# EPICS autosave request: iocBoot/ioc2/dbSave/23i_CS_Av_.req
%
% BURT Request File
%
% 23i:CS:Av:  Collimator (Monochromatic) slits, Vertical Aperture
%

file $(DIR)/assy.req ASSY=23i:CS:Av
23i:CS:Av:Invert
file $(DIR)/mtr1.req MTR1=23i:CS:mz1
file $(DIR)/mtr1.req MTR1=23i:CS:mz2
file $(DIR)/drv1.req DRV1=23i:CS:ZT
file $(DIR)/drv1.req DRV1=23i:CS:ZB
file $(DIR)/axs1.req AXS1=23i:CS:ZC
file $(DIR)/axs1.req AXS1=23i:CS:ZS
